// TIA Portal V20 export
ORGANIZATION_BLOCK "CyclicInterrupt"   // OB34, LAD, CyclicInterrupt
// stored: Namespace Unit1.Em6, SetENOAutomatically false
   VAR_INPUT
      Initial_Call : Bool;   // Initial call of this OB
      Event_Count : Int;   // Events discarded
   END_VAR
   VAR_TEMP
      tempIndex : Int;   // Index of EM in the array
   END_VAR
BEGIN

REGION Network 1: Call Equipment
END_REGION
END_ORGANIZATION_BLOCK
